FUNCTION_BLOCK XtsTrack IMPLEMENTS IXtsTrack
VAR_INPUT
	StateMachine : IPmlStateMachine;
	TmsSwitch : ITF_TmsSwitch;
END_VAR
VAR_OUTPUT
END_VAR
VAR
	_trackLength : MC_LREAL;
	_homePosition : MC_LREAL;
	HomeSpeed : MC_LREAL := 1000.0;
	mcCollisionGroup : CollisionGroup;
	XtsTrackHardware : XtsHardware;
	EnableSequence : XtsEnableSequence(mcCollisionGroup);
	DisableSequence : XtsDisableSequence(mcCollisionGroup);
	GroupStop : StopMoverGroup(mcCollisionGroup);
	State :(
        Init,                                           
		Ready,                                 
        Enabling,
		ActivateTracks,
		Enabled,
		Resetting,
		Idle,
		Running,
		Starting,
		Stop,
		Stopping,
		Disable,
		Disabling);  	
	i : DINT;
	AtHome: BOOL;
	_tracks : UDINT;
END_VAR
VAR_IN_OUT
	MoverArray : ARRAY[*] OF IMover;
END_VAR

XtsTrackHardware(Tracks := _tracks, TmsSwitch := TmsSwitch);
CASE State OF
	Init:
		IF XtsTrackHardware.XtsHardwareOK THEN
			GetTMSMoverInterface();
			State := Ready;
		END_IF
		
	Ready:
		IF StateMachine.GetCurrentState() = E_PMLState.ePMLState_Clearing THEN
			IF EnableSequence.Enable() THEN
				State := Enabling;
			END_IF	
		END_IF
		IF StateMachine.GetCurrentState() = E_PMLState.ePMLState_Aborting THEN		
			State := Disable;
		END_IF
		IF StateMachine.GetCurrentState() = E_PMLState.ePMLState_Stopping THEN		
			State := Stop;
		END_IF
		
	Enabling:
		IF EnableSequence.Done THEN
			State := ActivateTracks;
			StateMachine.SetStateComplete();
		END_IF
		
	ActivateTracks:
		IF ActivateTracksInMovers() THEN
			State := Enabled;
		END_IF
		
	Enabled:
		IF StateMachine.GetCurrentState() = E_PMLState.ePMLState_Resetting THEN
			IF MoverHomeSequence() THEN
				State := Resetting;
			END_IF
		END_IF
		IF StateMachine.GetCurrentState() = E_PMLState.ePMLState_Aborting THEN		
			State := Disable;
		END_IF
		IF StateMachine.GetCurrentState() = E_PMLState.ePMLState_Stopping THEN		
			State := Stop;
		END_IF
		
	Resetting:
		AtHome := TRUE;
		FOR i := LOWER_BOUND(MoverArray,1) TO UPPER_BOUND(MoverArray,1) DO
				AtHome := AtHome AND MoverArray[i].isStationary();
		END_FOR 
		IF AtHome THEN
			State := Idle;
			StateMachine.SetStateComplete();	
		END_IF
		
	Idle:	
		IF StateMachine.GetCurrentState() = E_PMLState.ePMLState_Starting THEN
			State := Starting;
		END_IF
		IF StateMachine.GetCurrentState() = E_PMLState.ePMLState_Aborting THEN		
			State := Disable;
		END_IF
		IF StateMachine.GetCurrentState() = E_PMLState.ePMLState_Stopping THEN		
			State := Stop;
		END_IF
		
	Starting:
		StateMachine.SetStateComplete();
		State := Running;
		
	Running:
		IF StateMachine.GetCurrentState() = E_PMLState.ePMLState_Aborting THEN		
			State := Disable;
		END_IF
		IF StateMachine.GetCurrentState() = E_PMLState.ePMLState_Stopping THEN		
			State := Stop;
		END_IF
		
	Stop:
		GroupStop.Execute();
		State := Stopping;
		
	Stopping:
		IF GroupStop.Done THEN
			State := Enabled;
			StateMachine.SetStateComplete();
		END_IF
		
	Disable:
		DisableSequence.Disable();
		State := Disabling;
		
	Disabling:
		IF DisableSequence.Done THEN
			State := Ready;
			StateMachine.SetStateComplete();
		END_IF
END_CASE

EnableSequence(arrMovers := MoverArray);
DisableSequence(arrMovers := MoverArray);
GroupStop();
mcCollisionGroup();

METHOD PUBLIC ActivateTracksInMovers : BOOL
VAR_INPUT
END_VAR
VAR
	iTmsMover : ITmsMover;
END_VAR
FOR i := 1 TO UPPER_BOUND(MoverArray,1) DO
	IF __QUERYINTERFACE(MoverArray[i],iTmsMover) THEN
		iTmsMover.ActivateTrack(newTrack := iTmsMover.ActiveTrack);
	END_IF
END_FOR
ActivateTracksInMovers := true;
END_METHOD

METHOD PUBLIC GetTMSMoverInterface : BOOL
VAR_INPUT
END_VAR
VAR
	iTmsMover : ITmsMover;
END_VAR
FOR i := 1 TO UPPER_BOUND(MoverArray,1) DO
	IF __QUERYINTERFACE(MoverArray[i],iTmsMover) THEN
		iTmsMover.SetMoverInterface(MoverInterface := XtsTrackHardware.GetMoverEnvInterface(DINT_TO_UINT(i)));
	END_IF
END_FOR
END_METHOD

PROPERTY PUBLIC HomePosition : mc_lreal
GET
HomePosition := _homePosition;
END_GET
SET
_homePosition := HomePosition;
END_SET
END_PROPERTY

METHOD PUBLIC MoverHomeSequence : BOOL
VAR_INPUT
END_VAR
FOR i := LOWER_BOUND(MoverArray,1) TO UPPER_BOUND(MoverArray,1) DO
	MoverArray[i].MoveTo(Position := _homePosition, Velocity := HomeSpeed, BackwardMove := FALSE);
END_FOR 
MoverHomeSequence := TRUE;
END_METHOD

PROPERTY PUBLIC TrackLength : mc_lreal
GET
TrackLength := _trackLength;
END_GET
SET // PUBLIC
_trackLength := TrackLength;
END_SET
END_PROPERTY

PROPERTY PUBLIC Tracks : UDINT
GET
Tracks := _tracks;
END_GET
SET
_tracks := Tracks;
END_SET
END_PROPERTY

END_FUNCTION_BLOCK

(* stored: Version 1.1.0.1, ProductVersion 3.1.4024.11
   POU XtsTrack: Id {9b564055-e4ef-49ec-91fa-4e16cb16a3f0}, SpecialFunc None
   Method ActivateTracksInMovers: Id {f07dde83-d085-4cf6-bf9b-a6e81e2388f6}
   Method GetTMSMoverInterface: Id {8a0ffa9f-0aa2-4c3c-a17d-9828995afbc3}
   Property HomePosition: Id {17d8d860-04e6-4fdc-9d29-4118d8eda955}
   Get Get: Id {620c6b86-3832-4e3f-9912-ef7e2a1a6514}
   Set Set: Id {f190637e-4d36-4143-baa6-9db775f41566}
   Method MoverHomeSequence: Id {75121f0d-c39e-4602-b6e8-ef3881ab6657}
   Property TrackLength: Id {4f244eb1-0239-423a-8574-4ccb93081483}
   Get Get: Id {962af0e5-68fc-457e-92c4-2ae643ddac5e}
   Set Set: Id {9d3b1cf5-ae4d-4af9-ab8c-ba44e55a4cc2}
   Property Tracks: Id {7741ef95-8846-4cc0-aa81-d8ac8ebba247}
   Get Get: Id {d2af4e1e-cc7b-4b07-b5c4-6cf6f6dda28f}
   Set Set: Id {bb7806ec-85ad-4f70-9606-95b8e7565462} *)
